// TIA Portal V16 export
// export: Created 2023-08-28T09:37:40.6819003Z, ExportSetting WithDefaults, DisplayName Totally Integrated Automation Portal, DisplayVersion V16 Update 6, DisplayName TIA Portal Version Control Interface, DisplayVersion V16 Update 2, DisplayName TIA Portal Openness, DisplayVersion V16 Update 6, DisplayName STEP 7 Professional, DisplayVersion V16 Update 6, DisplayName STEP 7 Safety, DisplayVersion V16, DisplayName WinCC Advanced, DisplayVersion V16 Update 6
FUNCTION_BLOCK "06_M_control without inverter"   // FB18, LAD
TITLE = Sterowania bez falownika
{ S7_Optimized_Access := 'TRUE' }
AUTHOR : rtecmer
VERSION : 0.1
// Sterowanie awaryjne układemw w wypadku awarii falownika.
// Sterowanie napędami z sieci. 
// Załączenie od sygnału  InputWarning_L_PID. jest to bit ustawiany przez regulator PID  wyliczany na podstawie wartości zadanej bar + wartość współczynnika .
// Wyłaczenie natępuje po osiągnięciu "Górnego progu tymczasowego". 
// Praca kompresorów z wyrównaniem liczników pracy.
// Jednocześnie pracuje tylko jeden kompresor.
// stored: AutoNumber true, IsIECCheckEnabled false, IsRetainMemResEnabled false, MemoryReserve 500, SetENOAutomatically false, UDAEnableTagReadback false
   VAR_INPUT
      IsReadyP1 : Bool;   // Gotowość pompy
      IsReadyP2 : Bool;   // Gotowość pompy
      IsReadyP3 : Bool;   // Gotowość pompy
      IsReadyP4 : Bool;
      IsMode_Auto : Bool;   // Tryb pracy Aut
      InputWarning_H_PID : Bool;   // Oszczerzenie górny limit
      InputWarning_L_PID : Bool;   // Oczszczerzenie dolny limit
      IsReady_Inverter : Bool;   // Gotowość falownika
      PV_max : Real;   // Wartość górnego progu ostrzegawczego
      Act_B3ciśnienie : Real;   // Aktualna wartość bar
      Rst_Driver_Max_presure : Bool;   // Znacznika awaryjnego wyłączenia od max ciśnienia napędu pracującego w trybie awaryjnym
   END_VAR
   VAR_OUTPUT
      CMD_A_Network_P1 : Bool;   // Bit startu pompyw trybie awaryjnym na soft-startcie
      CMD_A_Network_P2 : Bool := false;   // Bit startu pompyw trybie awaryjnym na soft-startcie
      CMD_A_Network_P3 : Bool := false;   // Bit startu pompyw trybie awaryjnym na soft-startcie
      CMD_A_Network_P4 : Bool := false;   // Bit startu pompyw trybie awaryjnym na soft-startcie
   END_VAR
   VAR
      stc_PV : Real := 0.2;   // Ustalona wartość pomniejszenia PV
   END_VAR
   VAR_TEMP
      set_Motor : Bool;   // pomocniczy bit ustawiający pompę
      tmp_PVmax : Real;   // Tymczasowa ustalona wartość progu górnego bar
   END_VAR
BEGIN

REGION Network 2: Górny próg tymczasowy
   // Wyliczenie górnego progu tymczasowego na potrzeby sterowania wyłączaniem pomp
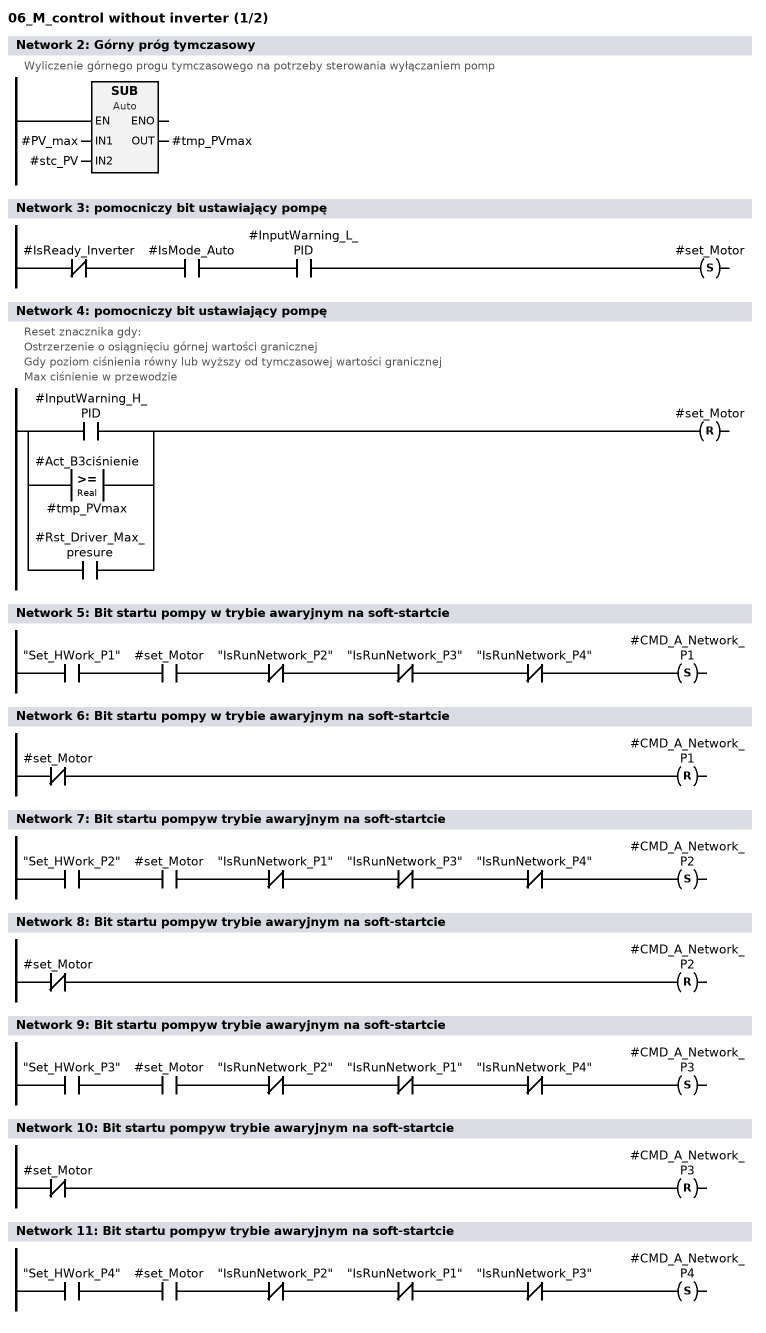
   RUNG wire#powerrail
      Sub(in1 := #PV_max, in2 := #stc_PV, out => #tmp_PVmax)
   END_RUNG
   // the same network as SCL:
   #tmp_PVmax := #PV_max - #stc_PV;
END_REGION

REGION Network 3: pomocniczy bit ustawiający pompę
   RUNG wire#powerrail
      I_Contact( #IsReady_Inverter )
      Contact( #IsMode_Auto )
      Contact( #InputWarning_L_PID )
      S_Coil( #set_Motor )
   END_RUNG
   // the same network as SCL:
   IF NOT #IsReady_Inverter AND #IsMode_Auto AND #InputWarning_L_PID THEN #set_Motor := TRUE; END_IF;
END_REGION

REGION Network 4: pomocniczy bit ustawiający pompę
   // Reset znacznika gdy:
   // Ostrzerzenie o osiągnięciu górnej wartości granicznej
   // Gdy poziom ciśnienia równy lub wyższy od tymczasowej wartości granicznej
   // Max ciśnienie w przewodzie
   RUNG wire#powerrail
      Contact( #InputWarning_H_PID )
      wire#w1
      R_Coil( #set_Motor )
   END_RUNG
   RUNG wire#powerrail
      { S7_Templates := "SrcType := Real" } GE_Contact(in1 := #Act_B3ciśnienie, in2 := #tmp_PVmax)
   END_RUNG wire#w1
   RUNG wire#powerrail
      Contact( #Rst_Driver_Max_presure )
   END_RUNG wire#w1
   // the same network as SCL:
   IF #InputWarning_H_PID OR (#Act_B3ciśnienie >= #tmp_PVmax) OR #Rst_Driver_Max_presure THEN
       #set_Motor := FALSE;
   END_IF;
END_REGION

REGION Network 5: Bit startu pompy w trybie awaryjnym na soft-startcie
   RUNG wire#powerrail
      Contact( "Set_HWork_P1" )
      Contact( #set_Motor )
      I_Contact( "IsRunNetwork_P2" )
      I_Contact( "IsRunNetwork_P3" )
      I_Contact( "IsRunNetwork_P4" )
      S_Coil( #CMD_A_Network_P1 )
   END_RUNG
   // the same network as SCL:
   IF "Set_HWork_P1" AND #set_Motor AND NOT "IsRunNetwork_P2" AND NOT "IsRunNetwork_P3" AND NOT "IsRunNetwork_P4" THEN
       #CMD_A_Network_P1 := TRUE;
   END_IF;
END_REGION

REGION Network 6: Bit startu pompy w trybie awaryjnym na soft-startcie
   RUNG wire#powerrail
      I_Contact( #set_Motor )
      R_Coil( #CMD_A_Network_P1 )
   END_RUNG
   // the same network as SCL:
   IF NOT #set_Motor THEN #CMD_A_Network_P1 := FALSE; END_IF;
END_REGION

REGION Network 7: Bit startu pompyw trybie awaryjnym na soft-startcie
   RUNG wire#powerrail
      Contact( "Set_HWork_P2" )
      Contact( #set_Motor )
      I_Contact( "IsRunNetwork_P1" )
      I_Contact( "IsRunNetwork_P3" )
      I_Contact( "IsRunNetwork_P4" )
      S_Coil( #CMD_A_Network_P2 )
   END_RUNG
   // the same network as SCL:
   IF "Set_HWork_P2" AND #set_Motor AND NOT "IsRunNetwork_P1" AND NOT "IsRunNetwork_P3" AND NOT "IsRunNetwork_P4" THEN
       #CMD_A_Network_P2 := TRUE;
   END_IF;
END_REGION

REGION Network 8: Bit startu pompyw trybie awaryjnym na soft-startcie
   RUNG wire#powerrail
      I_Contact( #set_Motor )
      R_Coil( #CMD_A_Network_P2 )
   END_RUNG
   // the same network as SCL:
   IF NOT #set_Motor THEN #CMD_A_Network_P2 := FALSE; END_IF;
END_REGION

REGION Network 9: Bit startu pompyw trybie awaryjnym na soft-startcie
   RUNG wire#powerrail
      Contact( "Set_HWork_P3" )
      Contact( #set_Motor )
      I_Contact( "IsRunNetwork_P2" )
      I_Contact( "IsRunNetwork_P1" )
      I_Contact( "IsRunNetwork_P4" )
      S_Coil( #CMD_A_Network_P3 )
   END_RUNG
   // the same network as SCL:
   IF "Set_HWork_P3" AND #set_Motor AND NOT "IsRunNetwork_P2" AND NOT "IsRunNetwork_P1" AND NOT "IsRunNetwork_P4" THEN
       #CMD_A_Network_P3 := TRUE;
   END_IF;
END_REGION

REGION Network 10: Bit startu pompyw trybie awaryjnym na soft-startcie
   RUNG wire#powerrail
      I_Contact( #set_Motor )
      R_Coil( #CMD_A_Network_P3 )
   END_RUNG
   // the same network as SCL:
   IF NOT #set_Motor THEN #CMD_A_Network_P3 := FALSE; END_IF;
END_REGION

REGION Network 11: Bit startu pompyw trybie awaryjnym na soft-startcie
   RUNG wire#powerrail
      Contact( "Set_HWork_P4" )
      Contact( #set_Motor )
      I_Contact( "IsRunNetwork_P2" )
      I_Contact( "IsRunNetwork_P1" )
      I_Contact( "IsRunNetwork_P3" )
      S_Coil( #CMD_A_Network_P4 )
   END_RUNG
   // the same network as SCL:
   IF "Set_HWork_P4" AND #set_Motor AND NOT "IsRunNetwork_P2" AND NOT "IsRunNetwork_P1" AND NOT "IsRunNetwork_P3" THEN
       #CMD_A_Network_P4 := TRUE;
   END_IF;
END_REGION

REGION Network 12: Bit startu pompyw trybie awaryjnym na soft-startcie
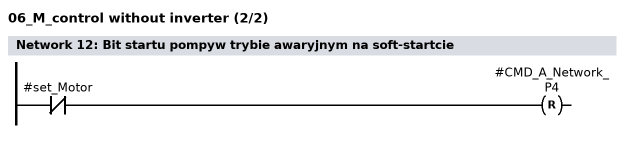
   RUNG wire#powerrail
      I_Contact( #set_Motor )
      R_Coil( #CMD_A_Network_P4 )
   END_RUNG
   // the same network as SCL:
   IF NOT #set_Motor THEN #CMD_A_Network_P4 := FALSE; END_IF;
END_REGION
END_FUNCTION_BLOCK
